FUNCTION_BLOCK CLNTRC_0_1 (* Wrapper for a CLIENT FB using the HTTP communciation protocol. Attempts to reconnect upon error. *)
  (* Standard: 61499-2 *)
  (* Version 0.0, 2017-09-05, 4DIAC-IDE, 4DIAC-Consortium *)
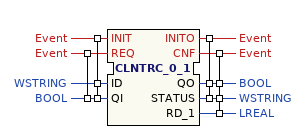
  EVENT_INPUT
    INIT WITH ID, QI; (* Initialization Request *)
    REQ WITH QI; (* Normal Execution Request *)
  END_EVENT
  EVENT_OUTPUT
    INITO WITH QO, STATUS; (* Initialization Confirm *)
    CNF WITH QO, STATUS, RD_1; (* Execution Confirmation *)
  END_EVENT
  VAR_INPUT
    ID : WSTRING; (* Connection Identifier *)
    QI : BOOL; (* Input event qualifier *)
  END_VAR
  VAR_OUTPUT
    QO : BOOL; (* Output event qualifier *)
    STATUS : WSTRING; (* Service Status *)
    RD_1 : LREAL; (* Received Data *)
  END_VAR
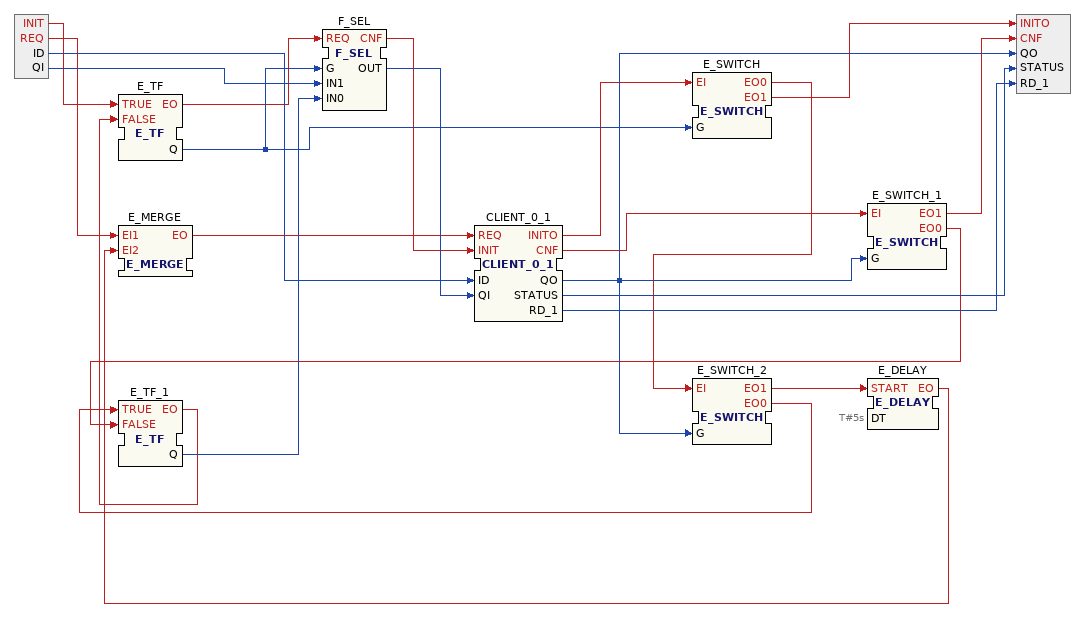
  FBS
    CLIENT_0_1 : CLIENT_0_1;
    E_TF : E_TF;
    E_SWITCH : E_SWITCH;
    E_MERGE : E_MERGE;
    E_SWITCH_1 : E_SWITCH;
    E_SWITCH_2 : E_SWITCH;
    E_DELAY : E_DELAY(DT := T#5s);
    E_TF_1 : E_TF;
    F_SEL : F_SEL;
  END_FBS
  EVENT_CONNECTIONS
    INIT TO E_TF.TRUE;
    CLIENT_0_1.INITO TO E_SWITCH.EI;
    REQ TO E_MERGE.EI1;
    E_SWITCH_1.EO1 TO CNF;
    E_SWITCH.EO0 TO E_SWITCH_2.EI;
    E_DELAY.EO TO E_MERGE.EI2;
    E_SWITCH_2.EO1 TO E_DELAY.START;
    CLIENT_0_1.CNF TO E_SWITCH_1.EI;
    E_MERGE.EO TO CLIENT_0_1.REQ;
    E_SWITCH.EO1 TO INITO;
    E_SWITCH_2.EO0 TO E_TF_1.TRUE;
    E_SWITCH_1.EO0 TO E_TF_1.FALSE;
    E_TF_1.EO TO E_TF.FALSE;
    E_TF.EO TO F_SEL.REQ;
    F_SEL.CNF TO CLIENT_0_1.INIT;
  END_CONNECTIONS
  DATA_CONNECTIONS
    ID TO CLIENT_0_1.ID;
    E_TF.Q TO E_SWITCH.G;
    CLIENT_0_1.QO TO E_SWITCH_1.G;
    CLIENT_0_1.QO TO E_SWITCH_2.G;
    CLIENT_0_1.STATUS TO STATUS;
    CLIENT_0_1.QO TO QO;
    CLIENT_0_1.RD_1 TO RD_1;
    E_TF.Q TO F_SEL.G;
    QI TO F_SEL.IN1;
    E_TF_1.Q TO F_SEL.IN0;
    F_SEL.OUT TO CLIENT_0_1.QI;
  END_CONNECTIONS
END_FUNCTION_BLOCK
